SUBAPPLICATION Uebung_010e (* SR und T-Flip-Flop mit 3x SoftKey (Softkey_IE, SK_RELEASED) mit GreenWhiteBackground am Toggle-SoftKey *)
  (* Standard: 61499-2; Description: Copyright (c) 2026 Meisterschulen am Ostbahnhof This program and the accompanying materials are made available under the terms of the Eclipse Public License 2.0 which is available at https://www.eclipse.org/legal/epl-2.0/ SPDX-License-Identifier: EPL-2.0 *)
  (* Version 1.0, 2026-09-02, Franz Höpfinger, Meisterschulen am Ostbahnhof, initial API and implementation and/or initial documentation *)
  PACKAGE Uebungen;
  IMPORT isobus::UT::io::Softkey::SoftKeyActivationCode::SK_RELEASED;
  IMPORT Uebungen::const::UT::DefaultPool::SoftKey_F1;
  IMPORT Uebungen::const::UT::DefaultPool::SoftKey_F2;
  IMPORT Uebungen::const::UT::DefaultPool::SoftKey_F3;
  IMPORT logiBUS::io::DQ::logiBUS_DO::Output_Q1;
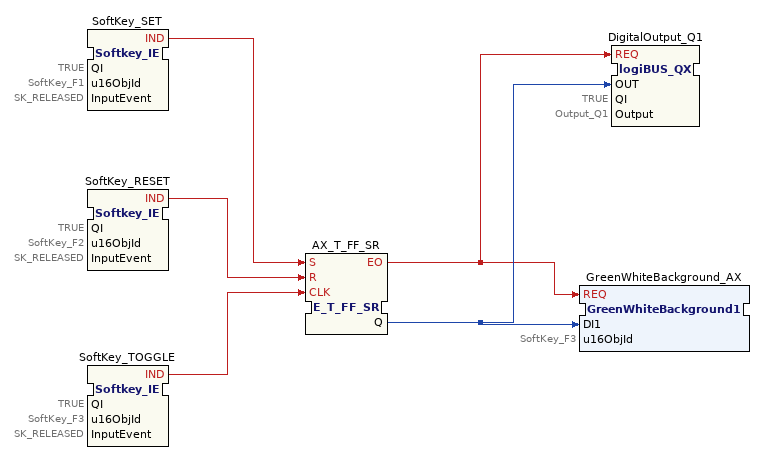
  FBS
    DigitalOutput_Q1 : logiBUS::io::DQ::logiBUS_QX(QI := TRUE, Output := Output_Q1);
    SoftKey_SET : isobus::UT::io::Softkey::Softkey_IE(QI := TRUE, u16ObjId := SoftKey_F1, InputEvent := SK_RELEASED);
    SoftKey_RESET : isobus::UT::io::Softkey::Softkey_IE(QI := TRUE, u16ObjId := SoftKey_F2, InputEvent := SK_RELEASED);
    SoftKey_TOGGLE : isobus::UT::io::Softkey::Softkey_IE(QI := TRUE, u16ObjId := SoftKey_F3, InputEvent := SK_RELEASED);
    AX_T_FF_SR : iec61499::events::E_T_FF_SR;
  END_FBS
  SUBAPPS
    GreenWhiteBackground_AX : MyLib::sys::GreenWhiteBackground1(u16ObjId := SoftKey_F3);
  END_SUBAPPS
  EVENT_CONNECTIONS
    SoftKey_SET.IND TO AX_T_FF_SR.S;
    SoftKey_RESET.IND TO AX_T_FF_SR.R;
    SoftKey_TOGGLE.IND TO AX_T_FF_SR.CLK;
    AX_T_FF_SR.EO TO DigitalOutput_Q1.REQ;
    AX_T_FF_SR.EO TO GreenWhiteBackground_AX.REQ;
  END_CONNECTIONS
  DATA_CONNECTIONS
    AX_T_FF_SR.Q TO DigitalOutput_Q1.OUT;
    AX_T_FF_SR.Q TO GreenWhiteBackground_AX.DI1;
  END_CONNECTIONS
END_SUBAPPLICATION
